TYPE "udtDbKomunikacja"
VERSION : 0.1
   STRUCT
      Trigger : Bool;
      NumerZlecenia : String[50];
      NumerOperacji : DInt;
      NumerPaletki : String[50];
      Stanowisko : String[50];
      Operator : String[50];
      CzasCykluMs : DInt;
      WynikQC : Bool;
      IloscWyprodukowanych : DInt;
      LiczbaWadliwych : DInt;
      KodPostoju : String[20];
   END_STRUCT;

END_TYPE

